(* IEC 61131-3 sources: brdkVision/export/brdkViImg/V5.21.0, 2 files *)

(* ---- brdkViImg.fun ---- *)
FUNCTION brdkViImg_freeMem : UDINT (*Function to free the memory buffer.*) (*$GROUP=User,$CAT=User,$GROUPICON=User.png,$CATICON=User.png*)
	VAR_INPUT
		pointer : UDINT; (*Pointer to the memory buffer.*)
	END_VAR
END_FUNCTION

FUNCTION brdkViImg_getPixel : USINT (*Function to return pixel value (0-255) at point x and y in image.*) (*$GROUP=User,$CAT=User,$GROUPICON=User.png,$CATICON=User.png*)
	VAR_INPUT
		x : INT; (*X coordinate in image.*)
		y : INT; (*Y coordinate in image.*)
		width : UDINT; (*Width of image.*)
		pSrc : REFERENCE TO USINT; (*Pointer to image data array.*)
	END_VAR
END_FUNCTION

FUNCTION brdkViImg_setPixel : BOOL (*Function to return pixel value (0-255) at point x and y in image.*) (*$GROUP=User,$CAT=User,$GROUPICON=User.png,$CATICON=User.png*)
	VAR_INPUT
		x : INT; (*X coordinate in image.*)
		y : INT; (*Y coordinate in image.*)
		width : UDINT; (*Width of image.*)
		pSrc : REFERENCE TO USINT; (*Pointer to image data array.*)
		color : USINT; (*Set color value*)
	END_VAR
END_FUNCTION

FUNCTION brdkViImg_getBmpImgInfo : BOOL (*Function to get BMP Image information. Returns True if BMP information is extracted. Returns False if no data is available or decoder encounters an error.*) (*$GROUP=User,$CAT=User,$GROUPICON=User.png,$CATICON=User.png*)
	VAR_INPUT
		pSrc : UDINT; (*Pointer to Image Data.*)
		len : UDINT; (*Size of the image.*)
	END_VAR
	VAR_IN_OUT
		pDest : brdkViImg_imageArray_typ; (*Pointer to brdkVIImg_imageArray where jpeg iformation is stored*)
	END_VAR
END_FUNCTION

FUNCTION brdkViImg_getJpegImgInfo : BOOL (*Function to get JPEG Image information. Returns True if JPEG information is extracted. Returns False if no data is available or decoder encounters an error.*) (*$GROUP=User,$CAT=User,$GROUPICON=User.png,$CATICON=User.png*)
	VAR_INPUT
		pSrc : UDINT; (*Pointer to Image Data.*)
		len : UDINT; (*Size of the image.*)
	END_VAR
	VAR_IN_OUT
		pDest : brdkViImg_imageArray_typ; (*Pointer to brdkVIImg_imageArray where jpeg iformation is stored*)
	END_VAR
END_FUNCTION

FUNCTION brdkViImg_base64Encode : BOOL (*Function to encode data to base64. Returns true on succesful encoding. Returns false on inter overflows. Returns %NULL on failure.*) (*$GROUP=User,$CAT=User,$GROUPICON=User.png,$CATICON=User.png*)
	VAR_INPUT
		pSrc : REFERENCE TO USINT; (*Pointer to data to be encoded.*)
		len : UDINT; (*Length of data to be encoded.*)
		pDest : REFERENCE TO USINT; (*Point to output location  where encoded data is stored*)
		maxDestLen : UDINT; (*Maximum length of encoded data.*)
	END_VAR
	VAR_IN_OUT
		pDestLen : UDINT; (* Pointer to UDINT where the size of the encoded data is stored*)
	END_VAR
END_FUNCTION

FUNCTION brdkViImg_base64Decode : BOOL (*Function to decode bae64 data type. Returns true on successful decoding. Returns false on unsuccesful decoding. Returns %NULL on failure.*) (*$GROUP=User,$CAT=User,$GROUPICON=User.png,$CATICON=User.png*)
	VAR_INPUT
		pSrc : REFERENCE TO USINT; (*Pointer data to be decoded.*)
		len : UDINT; (*Length of data to decoded.*)
		pDest : REFERENCE TO USINT; (*Pointer to output location of decoded data.*)
		maxDestLen : UDINT; (*Maximum length of decoded data.*)
	END_VAR
	VAR_IN_OUT
		pDestLen : UDINT; (* Pointer to UDINT where the size of the encoded data is stored*)
	END_VAR
END_FUNCTION

FUNCTION brdkViImg_bmpDecode : UDINT (*Function to decode BMP file format. Returns pData. Returns false if unexpected mask format and/or unexpected color space type. *) (*$GROUP=User,$CAT=User,$GROUPICON=User.png,$CATICON=User.png*)
	VAR_INPUT
		pSrc : UDINT; (*Pointer to source data.*)
		pDest : UDINT; (*Pointer to image data.*)
	END_VAR
	VAR_IN_OUT
		sizeMem : UDINT; (*Memory size.*)
		bmpHeader : brdkViImg_bmpHeader_typ; (*BMP header of type brdkViImg_bmpHeader.*)
		height : UDINT; (*Height of BMP image.*)
		width : UDINT; (*Width of BMP image.*)
		channels : USINT; (*Color channels of the image (1 if its grey scale)*)
	END_VAR
END_FUNCTION

{REDUND_UNREPLICABLE} FUNCTION_BLOCK brdkViImg_getImage (*Function block to download image from camera*) (*$GROUP=User,$CAT=User,$GROUPICON=User.png,$CATICON=User.png*)
	VAR_INPUT
		pMappLink : {REDUND_UNREPLICABLE} UDINT; (*Pointer to the vision component mapp variable fx. gCamera*)
		imageFormat : {REDUND_UNREPLICABLE} BRDKVIIMG_IMG_TYPE; (*Image format (BRDKVIIMG_IMG_TYPE_BMP or BRDKVIIMG_IMG_TYPE_JPG)*)
		simulateConfig : {REDUND_UNREPLICABLE} brdkViImg_getImageSimulate_typ; (*If true the image is decoded to an 2D array*)
		jpegQuality : {REDUND_UNREPLICABLE} USINT; (*Quality of the image (only JPEG)*)
		getImage : {REDUND_UNREPLICABLE} BOOL; (*Trigger download of image, (is automatically reset to false)*)
		enable : {REDUND_UNREPLICABLE} BOOL; (*Enable the function block.*)
		timeout : {REDUND_UNREPLICABLE} TIME := T#2000ms; (*Timeout will trigger a retry for download of  the image*)
	END_VAR
	VAR_OUTPUT
		pDest : {REDUND_UNREPLICABLE} UDINT; (*Pointer to memory containing the image*)
		destLen : {REDUND_UNREPLICABLE} UDINT; (*Size of the image*)
		initDone : {REDUND_UNREPLICABLE} BOOL; (*Initialization is done*)
		status : {REDUND_UNREPLICABLE} UINT; (*Status of the function block*)
	END_VAR
	VAR
		state : {REDUND_UNREPLICABLE} USINT;
		internal : {REDUND_UNREPLICABLE} brdkViImg_getImageInternal_typ;
		tmpStr1 : {REDUND_UNREPLICABLE} STRING[80];
	END_VAR
END_FUNCTION_BLOCK

{REDUND_UNREPLICABLE} FUNCTION_BLOCK brdkViImg_mappView (*Function block for loading an image from the memory buffer in mappView.*) (*$GROUP=User,$CAT=User,$GROUPICON=User.png,$CATICON=User.png*)
	VAR_INPUT
		enable : {REDUND_UNREPLICABLE} BOOL; (*Enable function block (will allocate/free memory)*)
		updateImage : {REDUND_UNREPLICABLE} BOOL; (*Trigger an update of the image (is automatically reset to false)*)
		simulateConfig : {REDUND_UNREPLICABLE} brdkViImg_getImageSimulate_typ; (*If true the image is decoded to an 2D array*)
		getImageArray : {REDUND_UNREPLICABLE} BOOL; (*If true the image is decoded to an 2D array*)
		imageFormat : {REDUND_UNREPLICABLE} BRDKVIIMG_IMG_TYPE; (*Image format (BRDKVIIMG_IMG_TYPE_BMP or BRDKVIIMG_IMG_TYPE_JPG)*)
		jpegQuality : {REDUND_UNREPLICABLE} USINT; (*Jpeg quality*)
		pMappLink : {REDUND_UNREPLICABLE} UDINT; (*Pointer to the vision component mapp variable fx. gCamera*)
		pSvgImage : {REDUND_UNREPLICABLE} UDINT; (*Pointer to the SVG string where data the image data should be added*)
		maxSvgImageLength : {REDUND_UNREPLICABLE} UDINT; (*Maximum lenght of the SVG string*)
		svgImagePosition : {REDUND_UNREPLICABLE} brdkViBase_2d_typ; (*Position of the image for the SVG string*)
		pImageArray : REFERENCE TO brdkViImg_imageArray_typ; (*Pointer to the image array structure where the decode image is stored along with information about it*)
		wsPort : {REDUND_UNREPLICABLE} UINT := 0; (*Websocket port number to accept connections from brdk Image Widgets (0=web socket is not used)*)
		timeout : {REDUND_UNREPLICABLE} UDINT := 6000; (*Timeout will trigger a retry for download of  the image*)
	END_VAR
	VAR_OUTPUT
		status : {REDUND_UNREPLICABLE} UINT; (*Status of the function block*)
		info : {REDUND_UNREPLICABLE} brdkViImg_mappViewInfo_typ; (*Execution information of the function block*)
		svgLength : {REDUND_UNREPLICABLE} UDINT; (*Actual lenght of the SVG string*)
		newSvgReady : {REDUND_UNREPLICABLE} BOOL; (*True when the SVG string have been updated*)
	END_VAR
	VAR
		internal : {REDUND_UNREPLICABLE} brdkViImg_mappViewInternal_typ;
	END_VAR
END_FUNCTION_BLOCK

{REDUND_UNREPLICABLE} FUNCTION_BLOCK brdkViImg_JpgEncode (*Function block to encode data to JPG format. *) (*$GROUP=User,$CAT=User,$GROUPICON=User.png,$CATICON=User.png*)
	VAR_INPUT
		execute : {REDUND_UNREPLICABLE} BOOL; (*Starts the JPG encoding.*)
		errorReset : {REDUND_UNREPLICABLE} BOOL; (*Reset error*)
		pSrc : {REDUND_UNREPLICABLE} UDINT; (*Source data of the JPG image.*)
		width : {REDUND_UNREPLICABLE} INT; (*Width of JPG Image.*)
		height : {REDUND_UNREPLICABLE} INT; (*Height of JPG Image.*)
		channels : {REDUND_UNREPLICABLE} INT; (*color channels (1 for grey scale image)*)
		quality : {REDUND_UNREPLICABLE} USINT; (*Quality of JPG Image. 1-99% (JPG is not lossless)*)
		pDest : {REDUND_UNREPLICABLE} UDINT; (*Pointer to destination data. (if zero memory will be allocated, based on the max_dest_size)*)
		max_dest_size : {REDUND_UNREPLICABLE} UDINT; (*Max dest size (JPG)*)
	END_VAR
	VAR_OUTPUT
		status : {REDUND_UNREPLICABLE} UINT; (*Status of the function block*)
		failedCnt : {REDUND_UNREPLICABLE} UDINT; (*Number of failed encoded of images*)
		done : {REDUND_UNREPLICABLE} BOOL; (*True  for one cycle when the encoding is done*)
		imgCnt : {REDUND_UNREPLICABLE} UDINT; (*Total number of encoded images*)
		size : {REDUND_UNREPLICABLE} UDINT; (*Output jpg size*)
	END_VAR
	VAR
		tmpDone : {REDUND_UNREPLICABLE} BOOL;
		taskIdent : {REDUND_UNREPLICABLE} UDINT;
		state : {REDUND_UNREPLICABLE} USINT;
		tick : {REDUND_UNREPLICABLE} USINT;
		tickOld : {REDUND_UNREPLICABLE} USINT;
		tonHeartbeat : {REDUND_UNREPLICABLE} TON;
		taskStatus : {REDUND_UNREPLICABLE} UDINT;
		name : {REDUND_UNREPLICABLE} STRING[10];
	END_VAR
END_FUNCTION_BLOCK

FUNCTION_BLOCK brdkViImg_JpgDecode (*Function block for decoding JPG image. Loads a JEPG image from a memory buffer or file. On return width/height will be set to image dimension, channels will be set to either 1 or 3.*) (*$GROUP=User,$CAT=User,$GROUPICON=User.png,$CATICON=User.png*)
	VAR_INPUT
		execute : {REDUND_UNREPLICABLE} BOOL; (*Starts the JPG decoding.*)
		errorReset : {REDUND_UNREPLICABLE} BOOL; (*Reset error*)
		pSrc : {REDUND_UNREPLICABLE} UDINT; (*Source data of the JPG image.*)
		len : {REDUND_UNREPLICABLE} UDINT; (*Extracts the size of the JPG image.*)
		max_dest_size : {REDUND_UNREPLICABLE} UDINT; (*Current size of the dest memory (if new is lower or equal the memory is reused)*)
		pDest : {REDUND_UNREPLICABLE} UDINT; (*Pointer to ouput decoded image data (if zero memory will be allocated based)*)
	END_VAR
	VAR_OUTPUT
		width : {REDUND_UNREPLICABLE} INT; (*Outputs width ofJPG image.*)
		height : {REDUND_UNREPLICABLE} INT; (*Outputs height of JPG Image.*)
		channels : {REDUND_UNREPLICABLE} INT; (*Color channels, 1 for greyscale or 3 for RGB colors.*)
		size : {REDUND_UNREPLICABLE} UDINT; (*Output image size*)
		status : {REDUND_UNREPLICABLE} UINT; (*Status of the function block*)
		done : {REDUND_UNREPLICABLE} BOOL; (*True  for one cycle when the decoding is done*)
		failedCnt : {REDUND_UNREPLICABLE} UDINT; (*Number of failed decodings of images*)
		imgCnt : {REDUND_UNREPLICABLE} UDINT; (*Total number of decoded images*)
	END_VAR
	VAR
		taskIdent : {REDUND_UNREPLICABLE} UDINT;
		state : {REDUND_UNREPLICABLE} USINT;
		tick : {REDUND_UNREPLICABLE} USINT;
		tickOld : {REDUND_UNREPLICABLE} USINT;
		tonHeartbeat : {REDUND_UNREPLICABLE} TON;
		tmpDone : {REDUND_UNREPLICABLE} BOOL;
		name : {REDUND_UNREPLICABLE} STRING[10];
		taskStatus : {REDUND_UNREPLICABLE} UDINT;
	END_VAR
END_FUNCTION_BLOCK

(* ---- Constants.var ---- *)
VAR CONSTANT
	ERR_BRDKVIIMG_BASE64_BUSY : UINT := 64001; (*Error occurring when base64 is busy.*)
	BRDKVIIMG_WS_BUFFER_SIZE : UDINT := 10000;
	BRDKVIIMG_WS_MAX_NUM_CLIENTS : UDINT := 10;
	ERR_BRDKVIIMG_SRC_LEN_IS_ZERO : UINT := 64011; (*Error occurring when source length is zero*)
	ERR_BRDKVIIMG_JPG_ENCODING_ERR : UINT := 64010; (*Error occurring when Jpeg encoding failed*)
	ERR_BRDKVIIMG_JPG_DECODING_ERR : UINT := 64009; (*Error occurring when Jpeg decoding failed*)
	ERR_BRDKVIIMG_MAX_LEN_IS_ZERO : UINT := 64008; (*Error occurring when max length is zero*)
	ERR_BRDKVIIMG_PSRC_IS_ZERO : UINT := 64007; (*Error occurring when pSrc is zero*)
	ERR_BRDKVIIMG_CHANNELS_IS_ZERO : UINT := 64006; (*Error occurring when channels is zero*)
	ERR_BRDKVIIMG_HEIGHT_IS_ZERO : UINT := 64005; (*Error occurring when height is zero*)
	ERR_BRDKVIIMG_WIDHT_IS_ZERO : UINT := 64004; (*Error occurring when width is zero*)
	ERR_BRDKVIIMG_SVG_LEN_TOO_SHORT : UINT := 64003; (*Error occurring when the SVG string supplied as input is not long enough*)
	ERR_BRDKVIIMG_NO_SIM_PFILE : UINT := 64002; (*Error occurring when no pFile pointer is supplied for simulation*)
	ERR_BRDKVIIMG_NO_IMAGE : UINT := 64000; (*Error occurring when no image is available*)
END_VAR
